FUNCTION_BLOCK FB_GetPrinterParameters
VAR_INPUT
	in_stNciToPlc: NCTOPLC_NCICHANNEL_REF;;
END_VAR
VAR_OUTPUT
	extruderValue: LREAL;
	extruderSpeed: LREAL;
END_VAR
VAR
	hParam: DINT;
	printerSpeed: LREAL;
END_VAR

hParam := ItpGetHParam( in_stNciToPlc );
extruderValue := (DINT_TO_LREAL (hParam)/100000);
printerSpeed := ItpGetSetPathVelocity( in_stNciToPlc );
extruderSpeed := (printerSpeed * 0.08);

IF extruderSpeed = 0  THEN // voorkomt dat de absolute commando een foutmeleding geeft
		extruderSpeed:= 0.01;
END_IF

END_FUNCTION_BLOCK

(* stored: Version 1.1.0.1, ProductVersion 3.1.4024.9
   POU FB_GetPrinterParameters: Id {07c56d90-d37b-4fab-887f-e05cc331526b}, SpecialFunc None *)
